# EPICS substitutions: utcaApp/Db/orbit_intlk.substitutions
file db/scan_task.template {
    {}
}

file db/orbit_intlk.template {
    {}
}
